// Mitsubishi GX Works2 project: plc-group4   PLC: FX3G

// global labels: Global1
VAR_GLOBAL
  start_day AT X007 : BOOL;
  input_chocolate AT D1100 : REAL;
  input_nuts AT D1300 : REAL;
  amount_nuts AT D1400 : REAL;
  input_pistachio AT D1500 : REAL;
  amount_pistachio AT D1600 : REAL;
  input_kadaif AT D1700 : REAL;
  amount_kadaif AT D1800 : REAL;
  workday_light AT Y007 : BOOL;
  lack_of_matirial AT M0 : BOOL;
  finish_day AT X005 : BOOL;
  start_chocolate_prepare AT X001 : BOOL;
  chocolate_check AT M1 : BOOL;
END_VAR
VAR_GLOBAL CONSTANT
  chocolate_for_init : REAL := 400.0;
  nuts_for_init : REAL := 100.0;
END_VAR
VAR_GLOBAL
  nuts_check AT M2 : BOOL;
  chocolate_ready_packs AT D7800 : REAL;
END_VAR
VAR_GLOBAL CONSTANT
  pistachio_for_init : REAL := 120.0;
END_VAR
VAR_GLOBAL
  pistachio_check AT M3 : BOOL;
END_VAR
VAR_GLOBAL CONSTANT
  kadaif_for_init : REAL := 60;
END_VAR
VAR_GLOBAL
  kadaif_check AT M4 : BOOL;
  chocolate_prepare_available AT M5 : BOOL;
  chocolate_melt_container AT D1210 : REAL;
  temperature_sensor AT X002 : BOOL;
  finish_trans_chocolate AT M6 : BOOL;
  finish_melting_process AT M7 : BOOL;
  mold_sensor AT X003 : BOOL;
  casting_light AT Y002 : BOOL;
  chocolate_molds AT D1900 : REAL;
  finish_casting AT M8 : BOOL;
  TC_casting AT TC1 : BOOL;
END_VAR
VAR_GLOBAL CONSTANT
  timer_casting : INT := 40;
END_VAR
VAR_GLOBAL
  check_light AT TS1 : BOOL;
  amount_chocolate1 AT D1240 : REAL;
END_VAR
VAR_GLOBAL CONSTANT
  starter_day : INT;
  melting_chocolate_amount : REAL := 400.0;
END_VAR
VAR_GLOBAL
  finish_move_chocolate AT M9 : BOOL;
  melting_light AT Y001 : BOOL;
  start_cream_preapre AT X004 : BOOL;
  analog_input1 AT D8280 : INT;
END_VAR
VAR_GLOBAL CONSTANT
  divide_int_num : REAL := 400;
END_VAR
VAR_GLOBAL
  save_analog_val AT D7900 : REAL;
  dubai_chocolate AT D7900 : REAL;
END_VAR
VAR_GLOBAL CONSTANT
  dubai_creame : REAL := 6;
END_VAR
VAR_GLOBAL
  select_dubai AT M10 : BOOL;
  nuts_chocolate AT D7900 : REAL;
END_VAR
VAR_GLOBAL CONSTANT
  nuts_creame : REAL := 5;
END_VAR
VAR_GLOBAL
  select_nuts AT M11 : BOOL;
END_VAR
VAR_GLOBAL CONSTANT
  nuts_to_dubai : REAL := 20;
END_VAR
VAR_GLOBAL
  cream_container AT D2000 : REAL;
END_VAR
VAR_GLOBAL CONSTANT
  pistachio_to_dubai : REAL := 120.0;
END_VAR
VAR_GLOBAL
  gta AT M12 : BOOL;
END_VAR
VAR_GLOBAL CONSTANT
  kadaif_to_dubai : REAL := 60;
  nuts_to_mix : REAL := 100;
  pistachio_to_mix : REAL := 100;
  ingredient_to_cream : REAL := 200;
END_VAR
VAR_GLOBAL
  start_timer AT M13 : BOOL;
  tc_cream_light_1 AT TC2 : BOOL;
END_VAR
VAR_GLOBAL CONSTANT
  timer_cream : INT := 10;
END_VAR
VAR_GLOBAL
  ts_cream_light AT TS2 : BOOL;
  cream_lightning_1 AT Y003 : BOOL;
  ts_cream_light2 AT TS3 : BOOL;
  cream_lightning_2 AT Y004 : BOOL;
  tc_cream_light_2 AT TC3 : BOOL;
  tc_cream AT TC4 : BOOL;
END_VAR
VAR_GLOBAL CONSTANT
  time_light_cream : INT := 50;
END_VAR
VAR_GLOBAL
  ts_cream_finish AT TS4 : BOOL;
  cream_finish AT M14 : BOOL;
  finish_select_cream AT M15 : BOOL;
  finish_cream AT M16 : BOOL;
  start_fridge_molds AT X006 : BOOL;
  tc_fridge AT TC5 : BOOL;
END_VAR
VAR_GLOBAL CONSTANT
  timer_fridge : INT := 30;
END_VAR
VAR_GLOBAL
  ts_fridge AT TS5 : BOOL;
  fridge_lightning AT Y006 : BOOL;
  finish_fridge AT M8 : BOOL;
  one_packing_unit AT X000 : BOOL;
  cc1 AT CC1 : BOOL;
END_VAR
VAR_GLOBAL CONSTANT
  one_mold : INT := 1;
END_VAR
VAR_GLOBAL
  cc2 AT CC2 : BOOL;
END_VAR
VAR_GLOBAL CONSTANT
  four_mold : INT := 4;
END_VAR
VAR_GLOBAL
  cs1 AT CS1 : BOOL;
  last_in_pack AT CS2 : BOOL;
  cs2 AT CS2 : BOOL;
  packing_in_process AT Y005 : BOOL;
  packing_end AT M18 : BOOL;
END_VAR
VAR_GLOBAL CONSTANT
  add_one : REAL := 1;
END_VAR
VAR_GLOBAL
  analog_light AT M19 : BOOL;
END_VAR
VAR_GLOBAL CONSTANT
  mul_num : INT := 400;
END_VAR
VAR_GLOBAL
  chocolate_ready_packs_number AT D2100 : REAL;
END_VAR
VAR_GLOBAL CONSTANT
  div_analog : REAL := 40;
END_VAR
VAR_GLOBAL
  analog_output AT D8282 : INT;
END_VAR
VAR_GLOBAL CONSTANT
  starter_day1 : REAL;
  more_iteration : INT;
  another_iteration : REAL;
END_VAR
VAR_GLOBAL
  init_all AT X011 : BOOL;
  init_all1 AT X010 : BOOL;
  finish_fridge1 AT M12 : BOOL;
END_VAR

// task Task_01 (event TRUE, interval 0, priority 31): POU_01

PROGRAM POU_01
(* structured ladder/FBD written out as ST: instructions are called as NAME(EN, inputs, outputs); _pN, _eN, _tN stand for wires *)
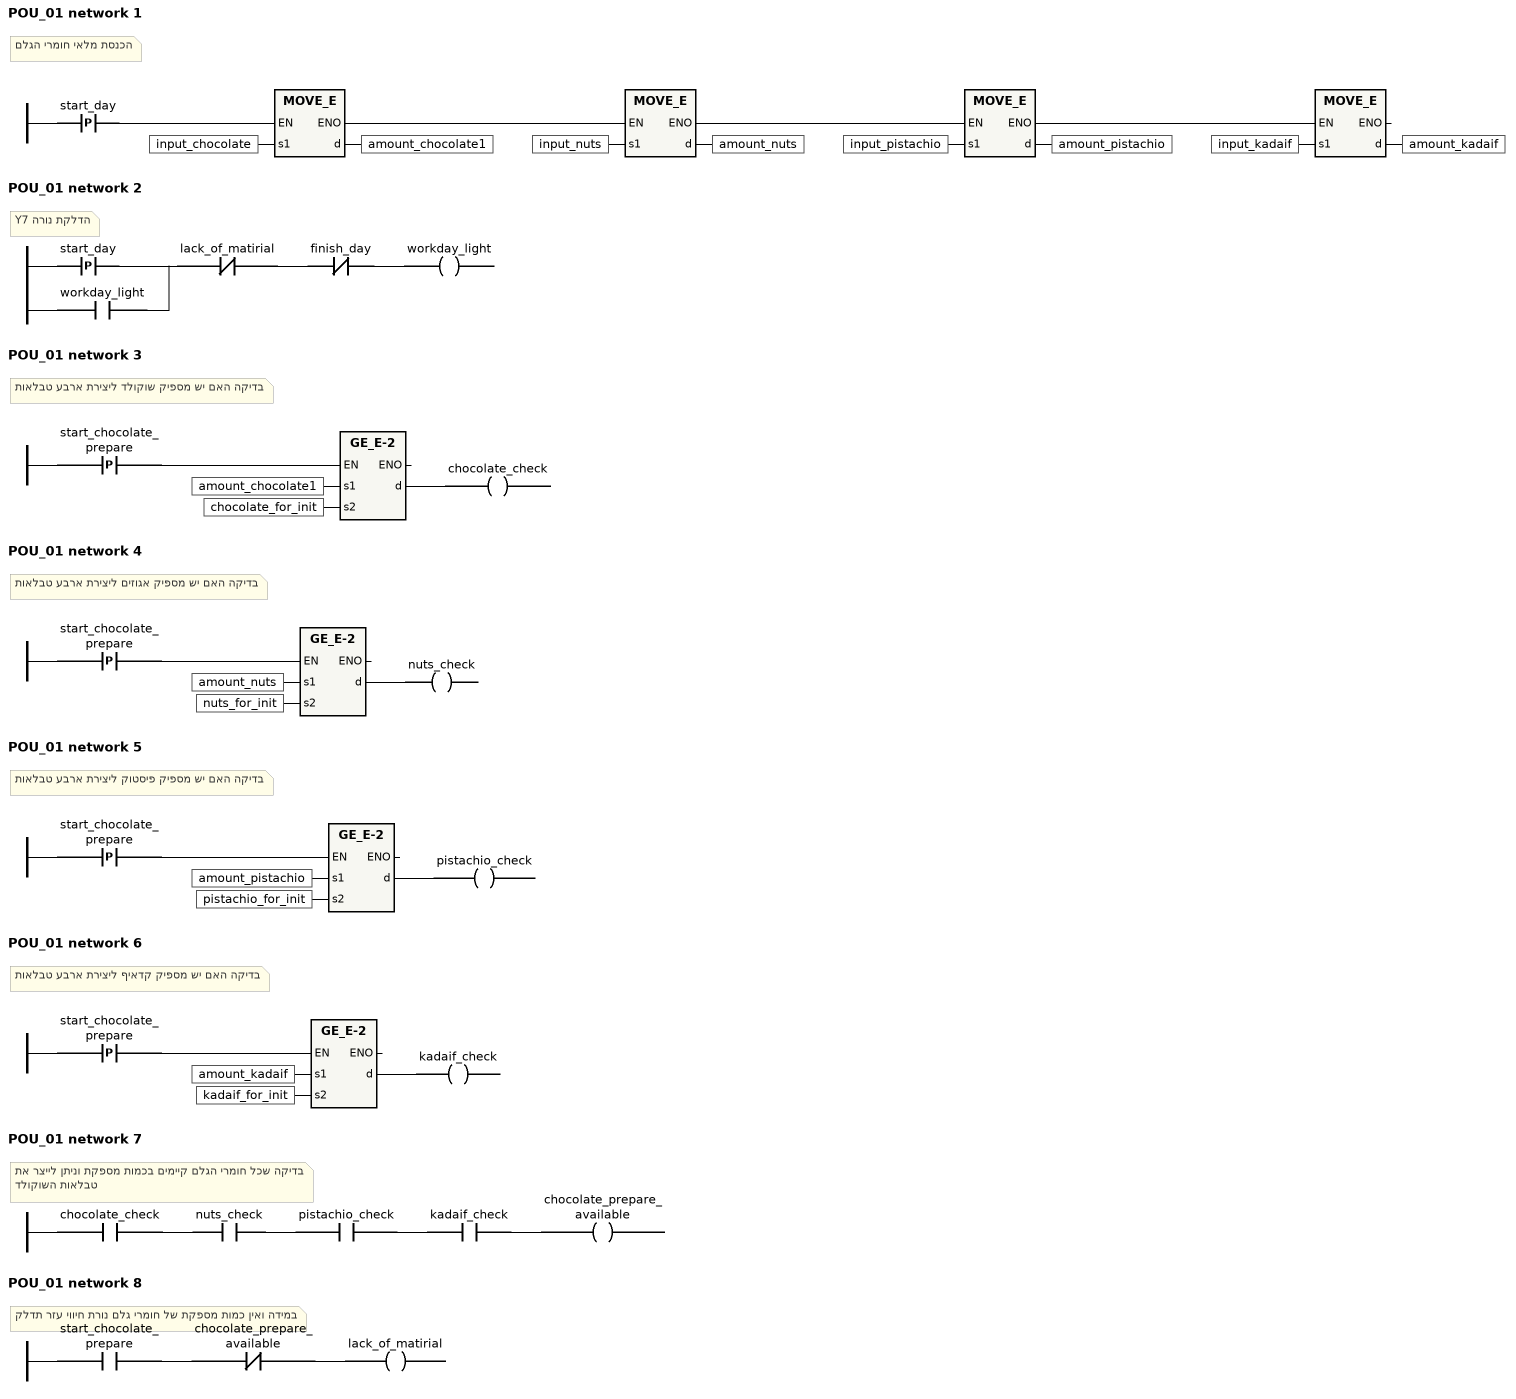
(* network 1 *)
(* הכנסת מלאי חומרי הגלם *)
_e1 := MOVE_E(LDP(TRUE, start_day), input_chocolate, amount_chocolate1);
_e2 := MOVE_E(_e1, input_nuts, amount_nuts);
_e3 := MOVE_E(_e2, input_pistachio, amount_pistachio);
MOVE_E(_e3, input_kadaif, amount_kadaif);
(* network 2 *)
(* Y7 הדלקת נורה *)
workday_light := ((LDP(TRUE, start_day) OR workday_light) AND NOT lack_of_matirial) AND NOT finish_day;
(* network 3 *)
(* בדיקה האם יש מספיק שוקולד ליצירת ארבע טבלאות *)
GE_E(LDP(TRUE, start_chocolate_prepare), amount_chocolate1, chocolate_for_init, _t1);
chocolate_check := _t1;
(* network 4 *)
(* בדיקה האם יש מספיק אגוזים ליצירת ארבע טבלאות *)
GE_E(LDP(TRUE, start_chocolate_prepare), amount_nuts, nuts_for_init, _t1);
nuts_check := _t1;
(* network 5 *)
(* בדיקה האם יש מספיק פיסטוק ליצירת ארבע טבלאות *)
GE_E(LDP(TRUE, start_chocolate_prepare), amount_pistachio, pistachio_for_init, _t1);
pistachio_check := _t1;
(* network 6 *)
(* בדיקה האם יש מספיק קדאיף ליצירת ארבע טבלאות *)
GE_E(LDP(TRUE, start_chocolate_prepare), amount_kadaif, kadaif_for_init, _t1);
kadaif_check := _t1;
(* network 7 *)
(* בדיקה שכל חומרי הגלם קיימים בכמות מספקת וניתן לייצר את טבלאות השוקולד *)
chocolate_prepare_available := chocolate_check AND nuts_check AND pistachio_check AND kadaif_check;
(* network 8 *)
(* במידה ואין כמות מספקת של חומרי גלם נורת חיווי עזר תדלק *)
lack_of_matirial := start_chocolate_prepare AND NOT chocolate_prepare_available;
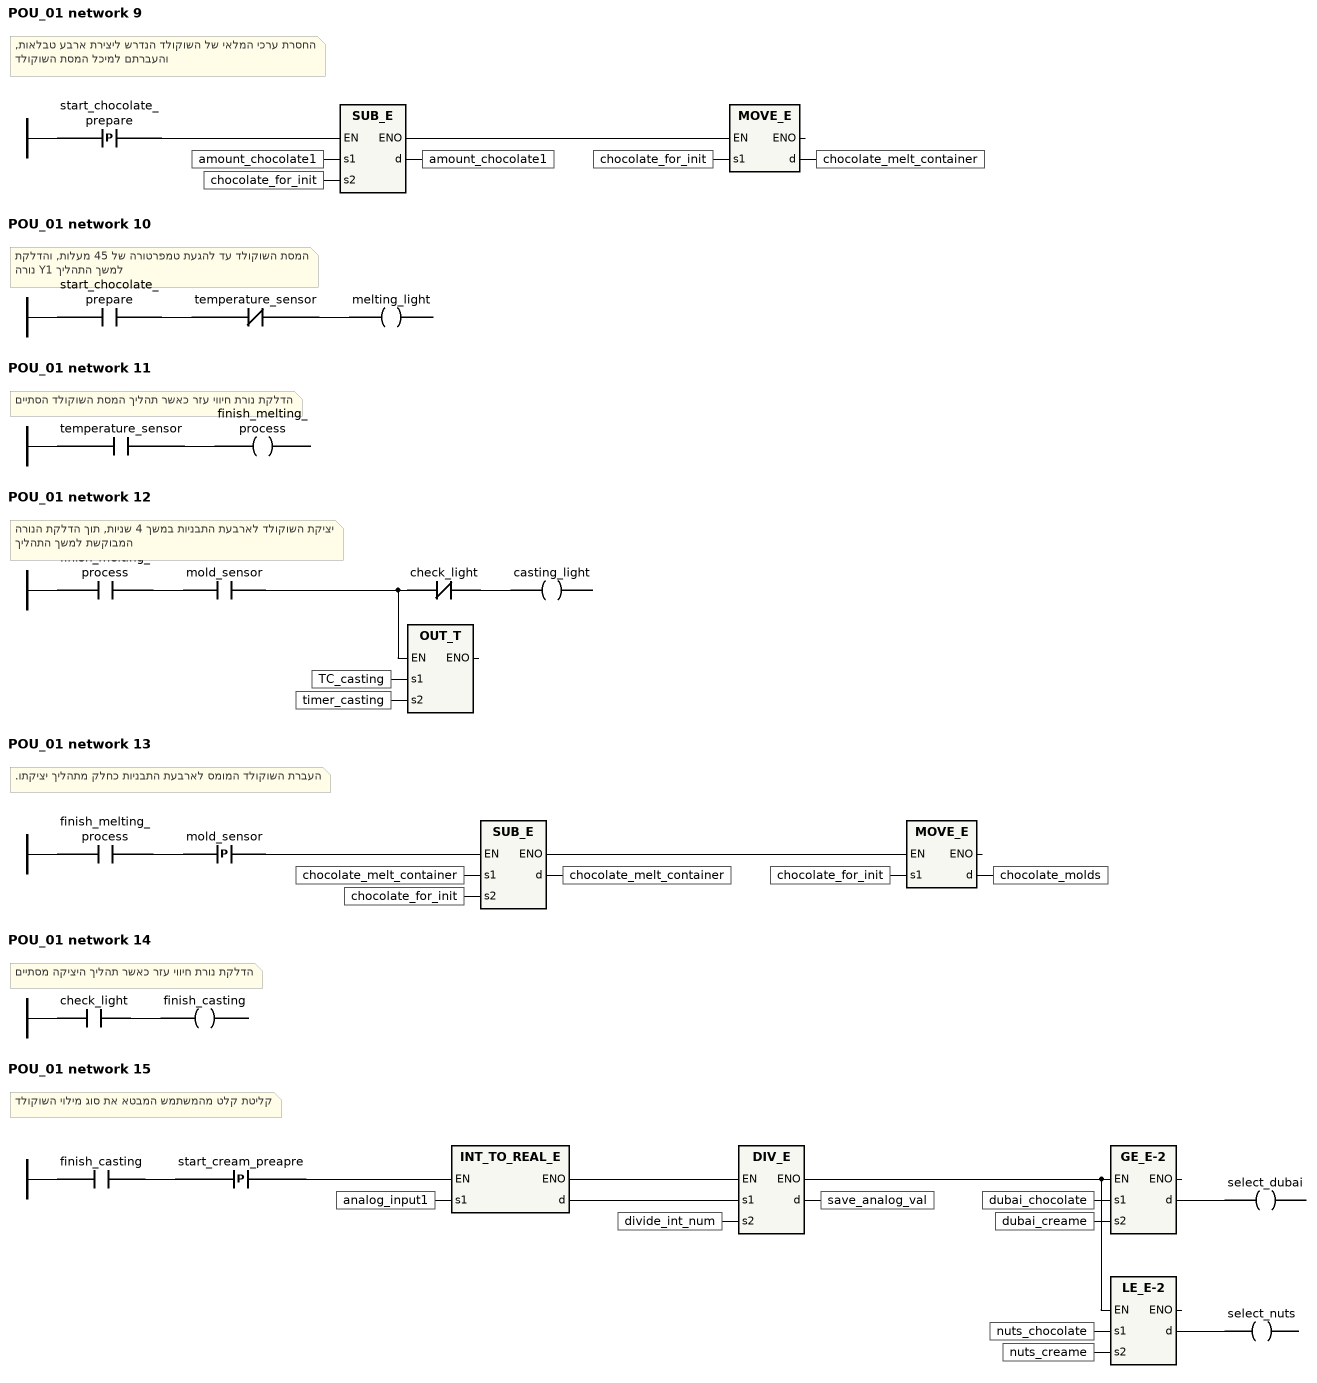
(* network 9 *)
(* החסרת ערכי המלאי של השוקולד הנדרש ליצירת ארבע טבלאות, והעברתם למיכל המסת השוקולד *)
_e1 := SUB_E(LDP(TRUE, start_chocolate_prepare), amount_chocolate1, chocolate_for_init, amount_chocolate1);
MOVE_E(_e1, chocolate_for_init, chocolate_melt_container);
(* network 10 *)
(* המסת השוקולד עד להגעת טמפרטורה של 45 מעלות, והדלקת  למשך התהליך Y1 נורה *)
melting_light := start_chocolate_prepare AND NOT temperature_sensor;
(* network 11 *)
(* הדלקת נורת חיווי עזר כאשר תהליך המסת השוקולד הסתיים *)
finish_melting_process := temperature_sensor;
(* network 12 *)
(* יציקת השוקולד לארבעת התבניות במשך 4 שניות, תוך הדלקת הנורה המבוקשת למשך התהליך *)
_p1 := finish_melting_process AND mold_sensor;
casting_light := _p1 AND NOT check_light;
OUT_T(_p1, TC_casting, timer_casting);
(* network 13 *)
(* העברת השוקולד המומס לארבעת התבניות כחלק מתהליך יציקתו. *)
_e1 := SUB_E(finish_melting_process AND LDP(TRUE, mold_sensor), chocolate_melt_container, chocolate_for_init, chocolate_melt_container);
MOVE_E(_e1, chocolate_for_init, chocolate_molds);
(* network 14 *)
(* הדלקת נורת חיווי עזר כאשר תהליך היציקה מסתיים *)
finish_casting := check_light;
(* network 15 *)
(* קליטת קלט מהמשתמש המבטא את סוג מילוי השוקולד *)
_e2 := INT_TO_REAL_E(finish_casting AND LDP(TRUE, start_cream_preapre), analog_input1, _t1);
_e3 := DIV_E(_e2, _t1, divide_int_num, save_analog_val);
GE_E(_e3, dubai_chocolate, dubai_creame, _t4);
select_dubai := _t4;
LE_E(_e3, nuts_chocolate, nuts_creame, _t5);
select_nuts := _t5;
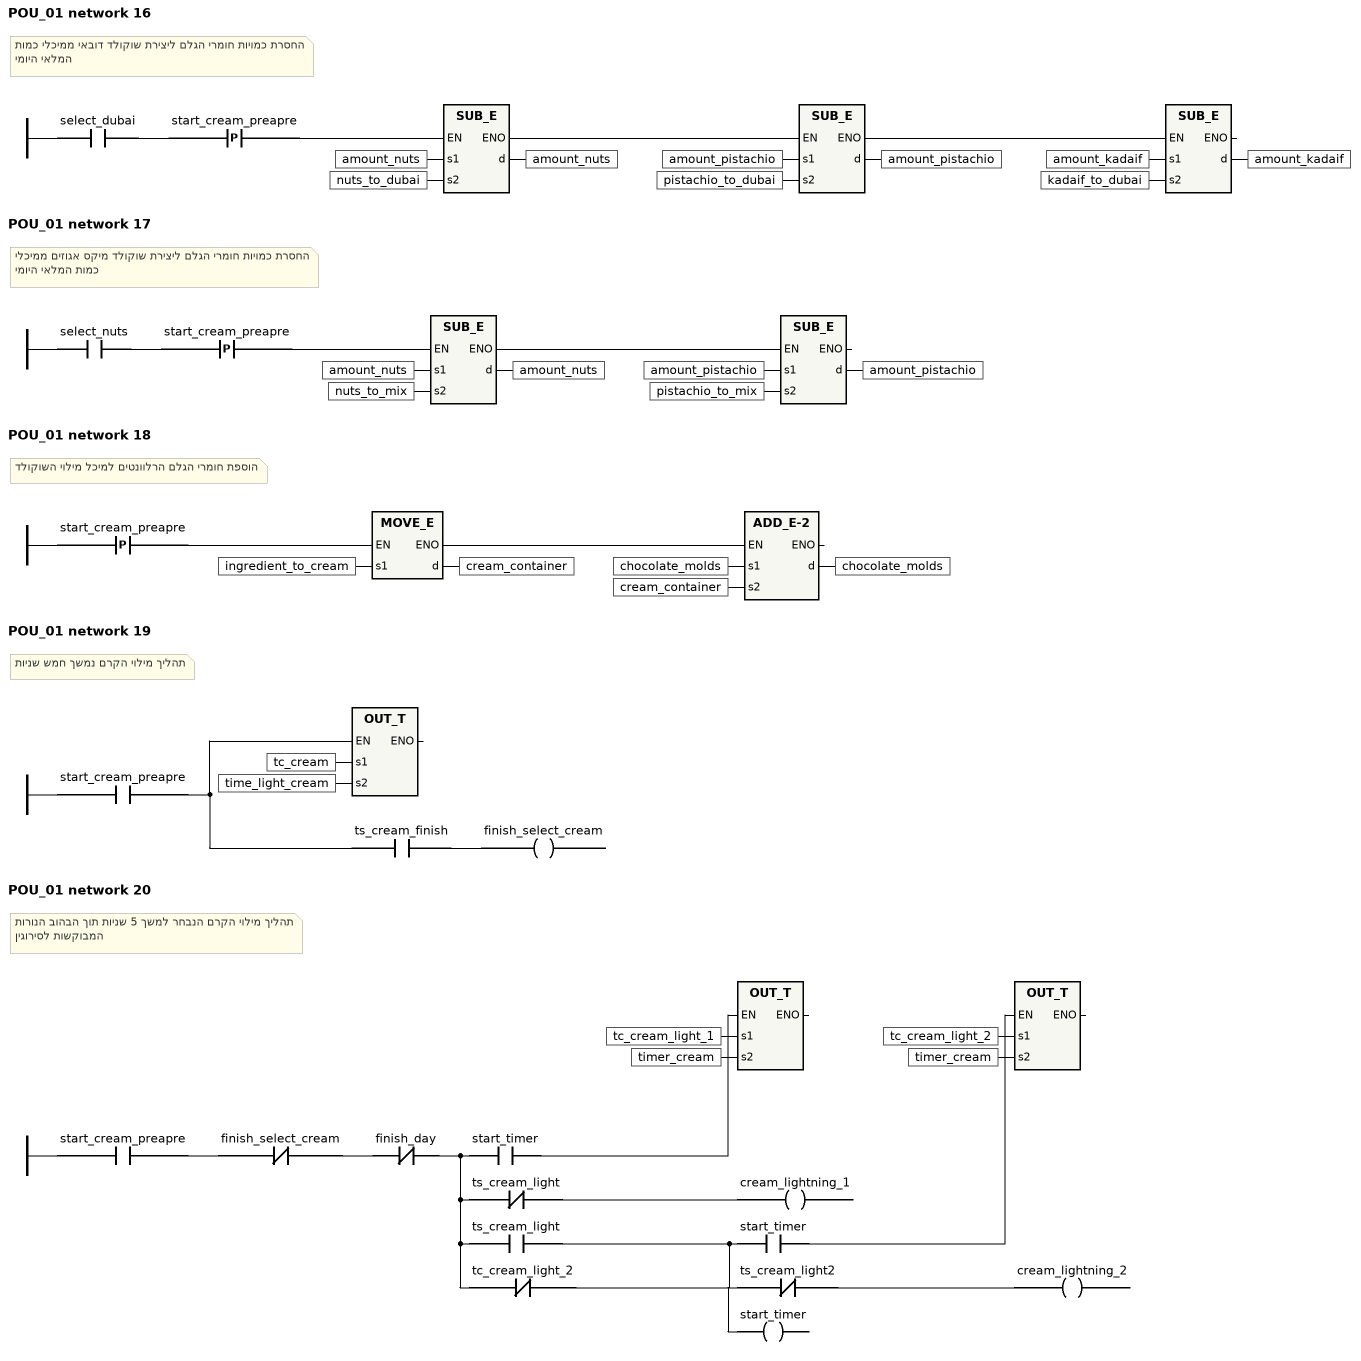
(* network 16 *)
(* החסרת כמויות חומרי הגלם ליצירת שוקולד דובאי ממיכלי כמות המלאי היומי *)
_e1 := SUB_E(select_dubai AND LDP(TRUE, start_cream_preapre), amount_nuts, nuts_to_dubai, amount_nuts);
_e2 := SUB_E(_e1, amount_pistachio, pistachio_to_dubai, amount_pistachio);
SUB_E(_e2, amount_kadaif, kadaif_to_dubai, amount_kadaif);
(* network 17 *)
(* החסרת כמויות חומרי הגלם ליצירת שוקולד מיקס אגוזים ממיכלי כמות המלאי היומי *)
_e1 := SUB_E(select_nuts AND LDP(TRUE, start_cream_preapre), amount_nuts, nuts_to_mix, amount_nuts);
SUB_E(_e1, amount_pistachio, pistachio_to_mix, amount_pistachio);
(* network 18 *)
(* הוספת חומרי הגלם הרלוונטים למיכל מילוי השוקולד *)
_e1 := MOVE_E(LDP(TRUE, start_cream_preapre), ingredient_to_cream, cream_container);
ADD_E(_e1, chocolate_molds, cream_container, chocolate_molds);
(* network 19 *)
(* תהליך מילוי הקרם נמשך חמש שניות *)
OUT_T(start_cream_preapre, tc_cream, time_light_cream);
finish_select_cream := start_cream_preapre AND ts_cream_finish;
(* network 20 *)
(* תהליך מילוי הקרם הנבחר למשך 5 שניות תוך הבהוב הנורות המבוקשות לסירוגין *)
_p1 := start_cream_preapre AND NOT finish_select_cream AND NOT finish_day;
OUT_T(_p1 AND start_timer, tc_cream_light_1, timer_cream);
cream_lightning_1 := _p1 AND NOT ts_cream_light;
_p2 := _p1 AND ts_cream_light;
OUT_T(_p2 AND start_timer, tc_cream_light_2, timer_cream);
cream_lightning_2 := _p2 AND NOT ts_cream_light2;
start_timer := _p1 AND NOT tc_cream_light_2;
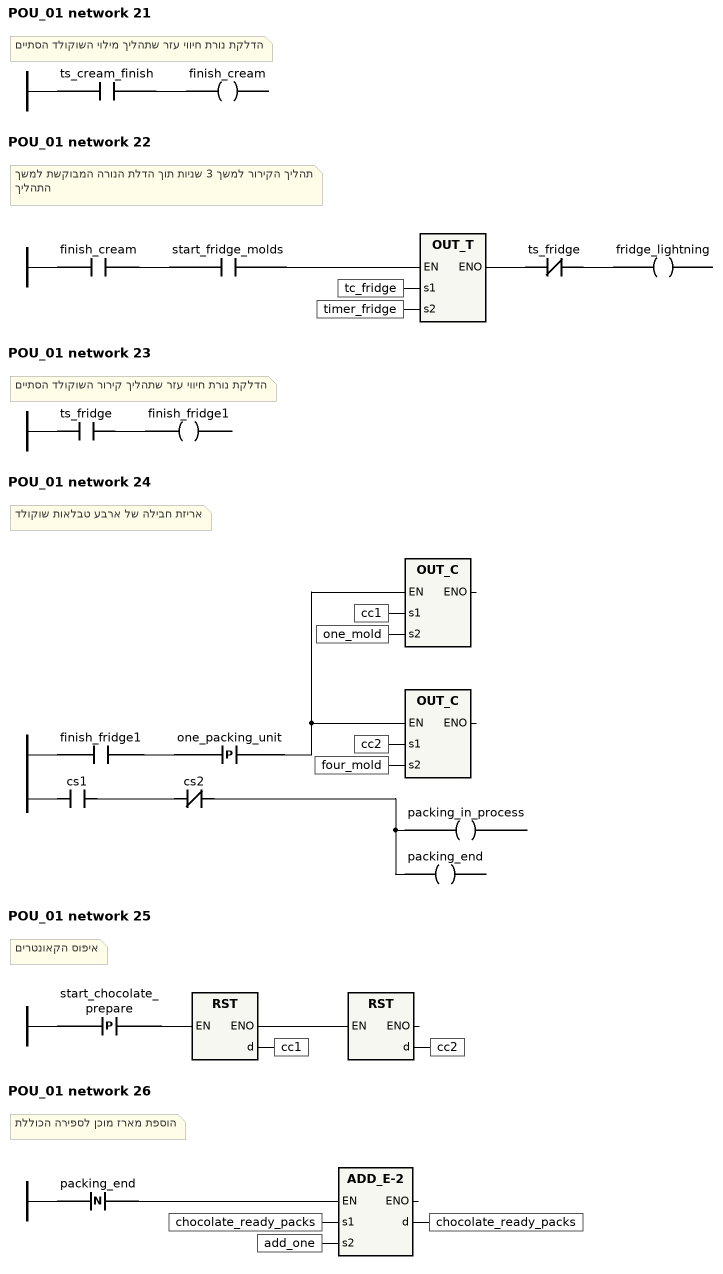
(* network 21 *)
(* הדלקת נורת חיווי עזר שתהליך מילוי השוקולד הסתיים *)
finish_cream := ts_cream_finish;
(* network 22 *)
(* תהליך הקירור למשך 3 שניות תוך הדלת הנורה המבוקשת למשך התהליך *)
_e1 := OUT_T(finish_cream AND start_fridge_molds, tc_fridge, timer_fridge);
fridge_lightning := _e1 AND NOT ts_fridge;
(* network 23 *)
(* הדלקת נורת חיווי עזר שתהליך קירור השוקולד הסתיים *)
finish_fridge1 := ts_fridge;
(* network 24 *)
(* אריזת חבילה של ארבע טבלאות שוקולד *)
_p1 := finish_fridge1 AND LDP(TRUE, one_packing_unit);
OUT_C(_p1, cc1, one_mold);
OUT_C(_p1, cc2, four_mold);
_p2 := cs1 AND NOT cs2;
packing_in_process := _p2;
packing_end := _p2;
(* network 25 *)
(* איפוס הקאונטרים *)
_e1 := RST(LDP(TRUE, start_chocolate_prepare), cc1);
RST(_e1, cc2);
(* network 26 *)
(* הוספת מארז מוכן לספירה הכוללת *)
ADD_E(LDF(TRUE, packing_end), chocolate_ready_packs, add_one, chocolate_ready_packs);
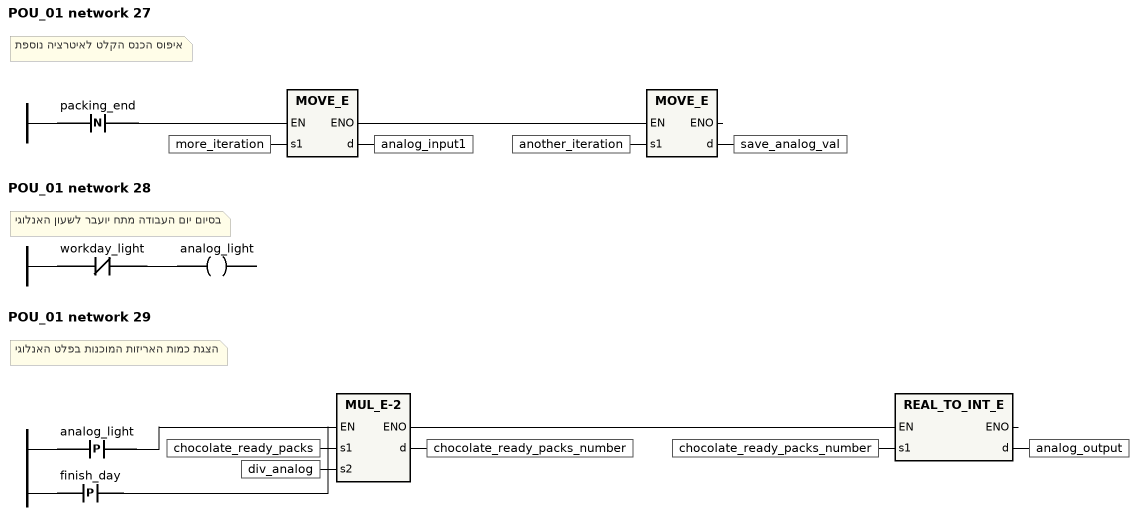
(* network 27 *)
(* איפוס הכנס הקלט לאיטרציה נוספת *)
_e1 := MOVE_E(LDF(TRUE, packing_end), more_iteration, analog_input1);
MOVE_E(_e1, another_iteration, save_analog_val);
(* network 28 *)
(* בסיום יום העבודה מתח יועבר לשעון האנלוגי *)
analog_light := NOT workday_light;
(* network 29 *)
(* הצגת כמות האריזות המוכנות בפלט האנלוגי *)
_e1 := MUL_E(LDP(TRUE, analog_light) OR LDP(TRUE, finish_day), chocolate_ready_packs, div_analog, chocolate_ready_packs_number);
REAL_TO_INT_E(_e1, chocolate_ready_packs_number, analog_output);
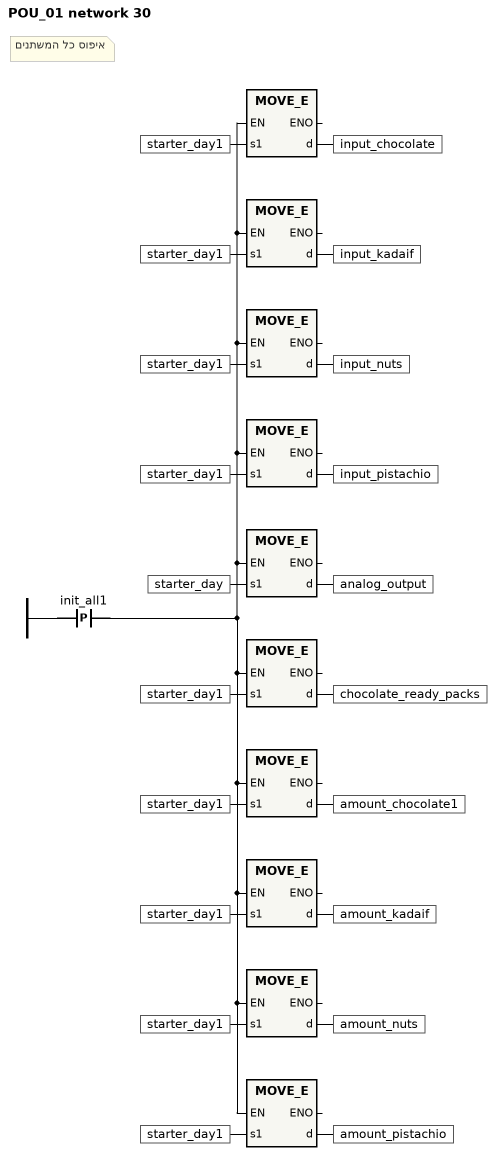
(* network 30 *)
(* איפוס כל המשתנים *)
_p1 := LDP(TRUE, init_all1);
MOVE_E(_p1, starter_day1, input_chocolate);
MOVE_E(_p1, starter_day1, input_kadaif);
MOVE_E(_p1, starter_day1, input_nuts);
MOVE_E(_p1, starter_day1, input_pistachio);
MOVE_E(_p1, starter_day, analog_output);
MOVE_E(_p1, starter_day1, chocolate_ready_packs);
MOVE_E(_p1, starter_day1, amount_chocolate1);
MOVE_E(_p1, starter_day1, amount_kadaif);
MOVE_E(_p1, starter_day1, amount_nuts);
MOVE_E(_p1, starter_day1, amount_pistachio);
END_PROGRAM
